(* Schneider Machine Expert - Basic project ProyekAkhir_Aradea Haikal Ikhwan_2106636880, file version 2.8.0.0 *)
(* ProjectInformations: Name=New project *)

HARDWARE
  Cpu 0: TM221M16R/G
  EthernetConfiguration: NetworkName=M221, IpAllocationMode=FixedAddress, IpAddress=0.0.0.0, SubnetMask=0.0.0.0
  SerialLineConfiguration: Baud=Baud19200, Parity=ParityEven, DataBits=DataBits8, StopBits=StopBits1, PhysicalMedium=PhysicalMediumRs485, TransmissionMode=TransmissionModeModbusRtu, SlaveId=1, Addressing=SlaveAddressing
  MastTask: UsePeriodScanMode=false, PeriodScan=100
  FastTask: Period=255
  CpuBehavior: StartingMode=StartAsPreviousState, AutoSaveRamOnEeprom=true, WatchdogPeriod=250

SYMBOLS  (address, symbol, comment, settings)
  %M0       S_VIS_BIRU
  %M1       DIFF_START_STOP
  %M2       MOV_X
  %M4       ITEM_DETECTED
  %M5       MULAI
  %M6       RESET
  %M7       STOP
  %M8       EMERGENCY_BUTTON
  %M11      DIFF_BIRU
  %M12      DIFF_HIJAU
  %M30      CONV
  %M31      CONV_1
  %M32      CONV_2
  %M33      CONV_3
  %M34      CONV_4
  %M35      CONV_5
  %M36      CONV_6
  %M37      CONV_7
  %M38      CONV_8
  %M39      CONV_9
  %M40      CONV_10
  %M41      PUSHER_BIRU
  %M42      PUSHER_HIJAU
  %M43      MOVE_X
  %M44      MOV_Z
  %M45      PNP_GRAB
  %M46      CONV_11
  %M47      LIGHT_START
  %M49      LIGHT_STOP
  %M120     MEM_1
  %M121     MEM_2
  %M122     MEM_3
  %M123     MEM_4
  %M124     MEM_5
  %M125     MEM_6
  %M126     MEM_7
  %M127     MEM_8
  %M128     MEM_9
  %TM0        [Preset=5, Base=OneHundredMilliSeconds]
  %TM1        [Preset=6, Base=OneHundredMilliSeconds]
  %TM2        [Preset=7, Base=OneHundredMilliSeconds]
  %TM3        [Preset=4, Base=OneHundredMilliSeconds]
  %TM4        [Preset=5, Base=OneHundredMilliSeconds]

POU POU  (* Pick and Place Conveyor Automatic Sorting System Based on it's Color *)
  (* SectionNumber=1 *)

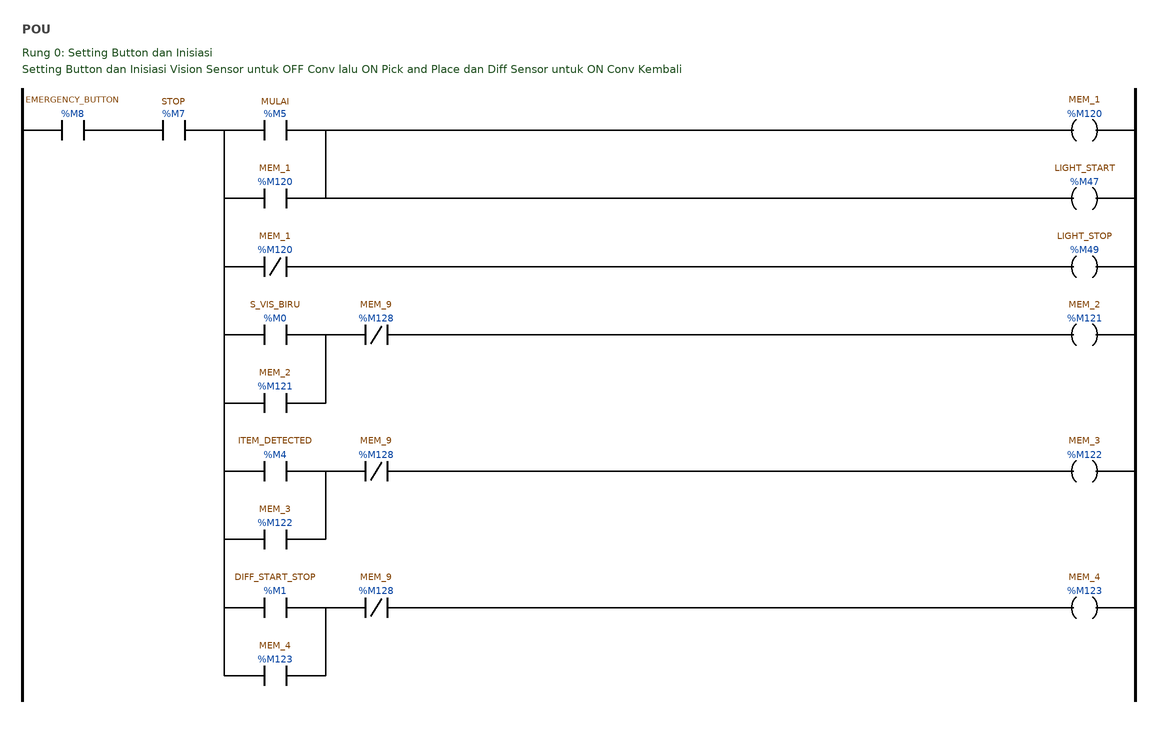

// Rung 0: Setting Button dan Inisiasi
// Setting Button dan Inisiasi Vision Sensor untuk OFF Conv lalu ON Pick and Place dan Diff Sensor untuk ON Conv Kembali
  LD %M8                  (* EMERGENCY_BUTTON *)
  AND %M7                 (* STOP *)
  MPS
  AND( %M5                (* MULAI *)
  OR %M120                (* MEM_1 *)
  )
  MPS
  ST %M120                (* MEM_1 *)
  MPP
  ST %M47                 (* LIGHT_START *)
  MRD
  ANDN %M120              (* MEM_1 *)
  ST %M49                 (* LIGHT_STOP *)
  MRD
  AND( %M0                (* S_VIS_BIRU *)
  OR %M121                (* MEM_2 *)
  )
  ANDN %M128              (* MEM_9 *)
  ST %M121                (* MEM_2 *)
  MRD
  AND( %M4                (* ITEM_DETECTED *)
  OR %M122                (* MEM_3 *)
  )
  ANDN %M128              (* MEM_9 *)
  ST %M122                (* MEM_3 *)
  MPP
  AND( %M1                (* DIFF_START_STOP *)
  OR %M123                (* MEM_4 *)
  )
  ANDN %M128              (* MEM_9 *)
  ST %M123                (* MEM_4 *)
  // as ST:
  //   _t1 := EMERGENCY_BUTTON AND STOP AND (MULAI OR MEM_1);
  //   MEM_1 := _t1;
  //   LIGHT_START := _t1;
  //   LIGHT_STOP := EMERGENCY_BUTTON AND STOP AND NOT MEM_1;
  //   MEM_2 := EMERGENCY_BUTTON AND STOP AND (S_VIS_BIRU OR MEM_2) AND NOT MEM_9;
  //   MEM_3 := EMERGENCY_BUTTON AND STOP AND (ITEM_DETECTED OR MEM_3) AND NOT MEM_9;
  //   MEM_4 := EMERGENCY_BUTTON AND STOP AND (DIFF_START_STOP OR MEM_4) AND NOT MEM_9;

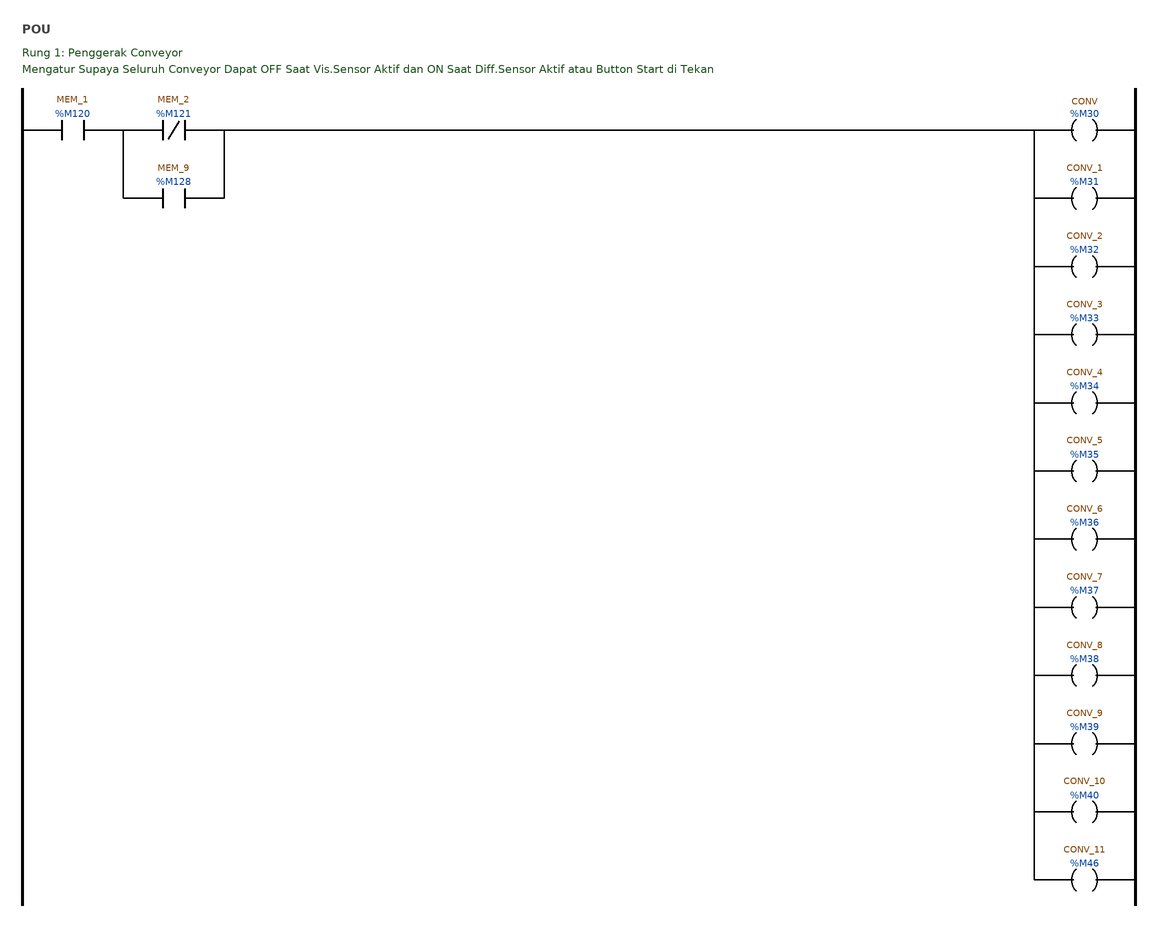

// Rung 1: Penggerak Conveyor
// Mengatur Supaya Seluruh Conveyor Dapat OFF Saat Vis.Sensor Aktif dan ON Saat Diff.Sensor Aktif atau Button Start di Tekan
  LD %M120                (* MEM_1 *)
  AND(N %M121             (* MEM_2 *)
  OR %M128                (* MEM_9 *)
  )
  ST %M30                 (* CONV *)
  ST %M31                 (* CONV_1 *)
  ST %M32                 (* CONV_2 *)
  ST %M33                 (* CONV_3 *)
  ST %M34                 (* CONV_4 *)
  ST %M35                 (* CONV_5 *)
  ST %M36                 (* CONV_6 *)
  ST %M37                 (* CONV_7 *)
  ST %M38                 (* CONV_8 *)
  ST %M39                 (* CONV_9 *)
  ST %M40                 (* CONV_10 *)
  ST %M46                 (* CONV_11 *)
  // as ST:
  //   CONV := MEM_1 AND (NOT MEM_2 OR MEM_9);
  //   CONV_1 := MEM_1 AND (NOT MEM_2 OR MEM_9);
  //   CONV_2 := MEM_1 AND (NOT MEM_2 OR MEM_9);
  //   CONV_3 := MEM_1 AND (NOT MEM_2 OR MEM_9);
  //   CONV_4 := MEM_1 AND (NOT MEM_2 OR MEM_9);
  //   CONV_5 := MEM_1 AND (NOT MEM_2 OR MEM_9);
  //   CONV_6 := MEM_1 AND (NOT MEM_2 OR MEM_9);
  //   CONV_7 := MEM_1 AND (NOT MEM_2 OR MEM_9);
  //   CONV_8 := MEM_1 AND (NOT MEM_2 OR MEM_9);
  //   CONV_9 := MEM_1 AND (NOT MEM_2 OR MEM_9);
  //   CONV_10 := MEM_1 AND (NOT MEM_2 OR MEM_9);
  //   CONV_11 := MEM_1 AND (NOT MEM_2 OR MEM_9);

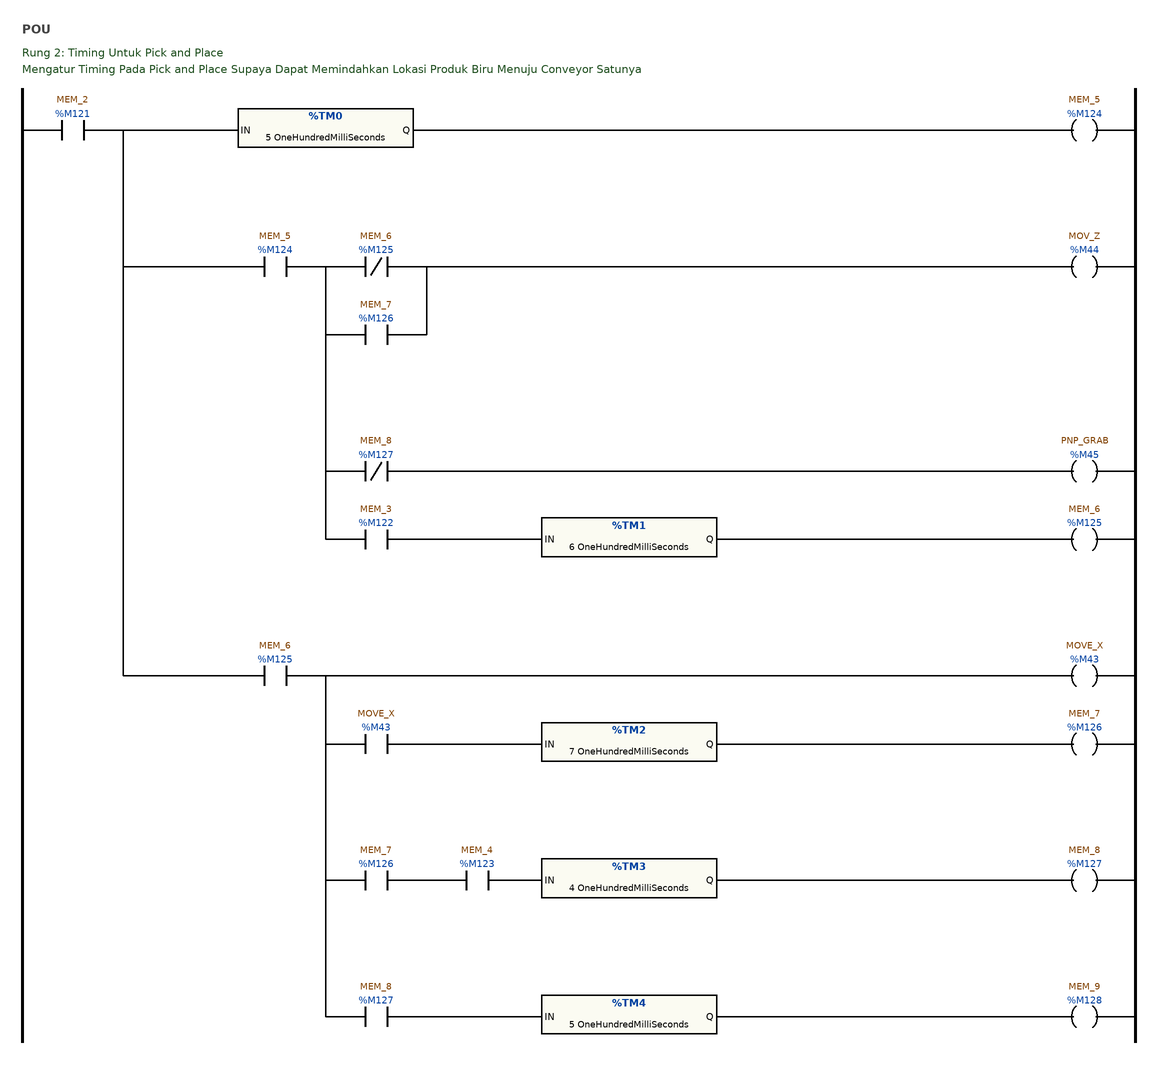

// Rung 2: Timing Untuk Pick and Place
// Mengatur Timing Pada Pick and Place Supaya Dapat Memindahkan Lokasi Produk Biru Menuju Conveyor Satunya
  LD 1
  MULTIFB
  LD 1
  AND %M121               (* MEM_2 *)
  ST %MW2009:X0
  BLK %TM0
  LD %MW2009:X0
  IN
  OUT_BLK
  LD Q
  ST %M124                (* MEM_5 *)
  END_BLK
  LD %MW2009:X0
  AND %M124               (* MEM_5 *)
  ST %MW2009:X1
  LD %MW2009:X1
  MPS
  AND(N %M125             (* MEM_6 *)
  OR %M126                (* MEM_7 *)
  )
  ST %M44                 (* MOV_Z *)
  MPP
  ANDN %M127              (* MEM_8 *)
  ST %M45                 (* PNP_GRAB *)
  BLK %TM1
  LD %MW2009:X1
  AND %M122               (* MEM_3 *)
  IN
  OUT_BLK
  LD Q
  ST %M125                (* MEM_6 *)
  END_BLK
  LD %MW2009:X0
  AND %M125               (* MEM_6 *)
  ST %MW2009:X2
  LD %MW2009:X2
  ST %M43                 (* MOVE_X *)
  BLK %TM2
  LD %MW2009:X2
  AND %M43                (* MOVE_X *)
  IN
  OUT_BLK
  LD Q
  ST %M126                (* MEM_7 *)
  END_BLK
  BLK %TM3
  LD %MW2009:X2
  AND %M126               (* MEM_7 *)
  AND %M123               (* MEM_4 *)
  IN
  OUT_BLK
  LD Q
  ST %M127                (* MEM_8 *)
  END_BLK
  BLK %TM4
  LD %MW2009:X2
  AND %M127               (* MEM_8 *)
  IN
  OUT_BLK
  LD Q
  ST %M128                (* MEM_9 *)
  END_BLK
  MULTIFB
  // as ST:
  //   %TM0(IN := MEM_2);
  //   MEM_5 := %TM0.Q;
  //   MOV_Z := MEM_2 AND MEM_5 AND (NOT MEM_6 OR MEM_7);
  //   PNP_GRAB := MEM_2 AND MEM_5 AND NOT MEM_8;
  //   %TM1(IN := MEM_2 AND MEM_5 AND MEM_3);
  //   MEM_6 := %TM1.Q;
  //   MOVE_X := MEM_2 AND MEM_6;
  //   %TM2(IN := MEM_2 AND MEM_6 AND MOVE_X);
  //   MEM_7 := %TM2.Q;
  //   %TM3(IN := MEM_2 AND MEM_6 AND MEM_7 AND MEM_4);
  //   MEM_8 := %TM3.Q;
  //   %TM4(IN := MEM_2 AND MEM_6 AND MEM_8);
  //   MEM_9 := %TM4.Q;

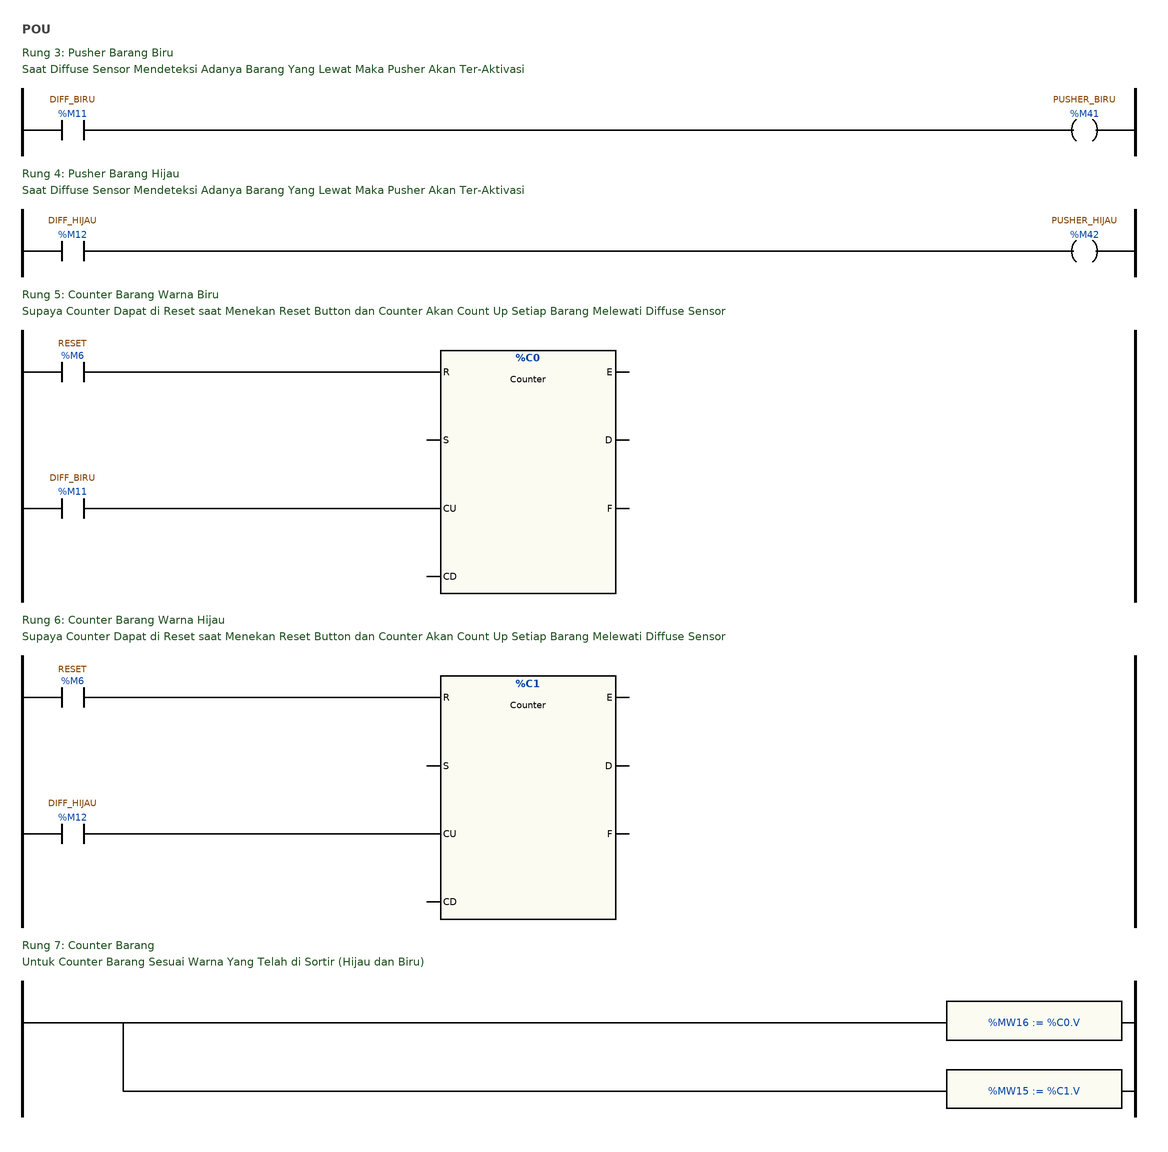

// Rung 3: Pusher Barang Biru
// Saat Diffuse Sensor Mendeteksi Adanya Barang Yang Lewat Maka Pusher Akan Ter-Aktivasi
  LD %M11                 (* DIFF_BIRU *)
  ST %M41                 (* PUSHER_BIRU *)
  // as ST:
  //   PUSHER_BIRU := DIFF_BIRU;

// Rung 4: Pusher Barang Hijau
// Saat Diffuse Sensor Mendeteksi Adanya Barang Yang Lewat Maka Pusher Akan Ter-Aktivasi
  LD %M12                 (* DIFF_HIJAU *)
  ST %M42                 (* PUSHER_HIJAU *)
  // as ST:
  //   PUSHER_HIJAU := DIFF_HIJAU;

// Rung 5: Counter Barang Warna Biru
// Supaya Counter Dapat di Reset saat Menekan Reset Button dan Counter Akan Count Up Setiap Barang Melewati Diffuse Sensor
  BLK %C0
  LD %M6                  (* RESET *)
  R
  LD %M11                 (* DIFF_BIRU *)
  CU
  END_BLK
  // as ST:
  //   %C0(R := RESET, CU := DIFF_BIRU);

// Rung 6: Counter Barang Warna Hijau
// Supaya Counter Dapat di Reset saat Menekan Reset Button dan Counter Akan Count Up Setiap Barang Melewati Diffuse Sensor
  BLK %C1
  LD %M6                  (* RESET *)
  R
  LD %M12                 (* DIFF_HIJAU *)
  CU
  END_BLK
  // as ST:
  //   %C1(R := RESET, CU := DIFF_HIJAU);

// Rung 7: Counter Barang
// Untuk Counter Barang Sesuai Warna Yang Telah di Sortir (Hijau dan Biru)
  LD 1
  [ %MW16 := %C0.V ]
  [ %MW15 := %C1.V ]
  // as ST:
  //   %MW16 := %C0.V;
  //   %MW15 := %C1.V;
